// TwinCAT 3 PLC project PLC1
// ProgramVersion: 3.1.4024.0
// libraries:
//   SPT Vision, * (Beckhoff Automation LLC)
//   Tc2_Standard, * (Beckhoff Automation GmbH)
//   Tc2_System, * (Beckhoff Automation GmbH)
//   Tc3_Module, * (Beckhoff Automation GmbH)
//   Tc3_Vision, * (Beckhoff Automation GmbH)
// project tree:
//   / GlobalTextList.TcGTLO, PlcTask.TcTTO (not stored), Visualization Manager.TcVMO (not stored)
//   POUs/ FB_ImageAquire.TcPOU (not stored), MAIN.TcPOU
//   VISUs/ V_Main.TcVIS (not stored)
// real-time tasks:
//   TASK VnTask ImgAcq (FileSource1): cycle T#10ms, priority 5, ADS port 351
//   TASK PlcTask1: cycle T#10ms, priority 20, ADS port 352

// ---- POUs/MAIN.TcPOU
PROGRAM MAIN
VAR
	Camera1 : FB_ImageAquire; 


	Playback : FB_ImageToVideo := (CameraName 			:= 'Camera1', 
							   	   JsonAttribute 		:= '{CreateVid : 1, CameraName: "Camera1"}', 
							   	   FramesPerSecond 		:= 10,
							   	   TimeBeforeEvent		:= T#7S,
								   TimeAfterEvent		:= T#3S,
								   VideoOutputDirectory := 'C:\Videos',
								   ReductionFactor 		:= 0.25,
								   Codec 				:= 'H264');

	TriggerEvent : BOOL;
END_VAR

Camera1.CyclicLogic();
IF Camera1.ImageAvailable THEN
	Playback.AddImage(ipImageIn := Camera1.Image);
END_IF

Playback.CyclicLogic();
IF TriggerEvent THEN
	TriggerEvent := FALSE;
	Playback.TriggerAlarmForVideoCapture();
END_IF

END_PROGRAM

// ---- GlobalTextList.TcGTLO
TEXTLIST GlobalTextList
  628 = 'Reset Playback'
  263 = 'Run Vision'
  459 = 'Trigger Video'
END_TEXTLIST
